// TIA Portal V19 export
TYPE "pulsante"
   STRUCT
      start : Bool;
      stop : Bool;
   END_STRUCT;
END_TYPE
